FUNCTION_BLOCK FB_System_BSp_795
VAR_INPUT
	Freigabe_auto			: BOOL;
	Freigabe_Deakt_auto		: BOOL;
	Betrieb_Anford_auto		: BOOL;

	Regelung_Modus_auto		: SINT;
	Regelung_Sollw_auto		: REAL;

	Temp_Netz_KW			: REAL; (*Temperatur kommt aus den Netzen; setzt sich zusammen aus Temperatur der Pufferspeicher, dem Betonspeicher und der Umgebungstemperatur*)
END_VAR
VAR_OUTPUT
	{attribute 'OPC.UA.DA' := '1'}Steuerung				: ST_System_BSp_Steuerung;		
	{attribute 'OPC.UA.DA' := '1'}Stellwert				: ST_System_BSp_Stellwert;		
	{attribute 'OPC.UA.DA' := '1'}Zustand					: ST_System_BSp_Zustand;	
	{attribute 'OPC.UA.DA' := '1'}Parameter				: ST_System_BSp_Parameter;		
END_VAR
VAR
	Stellventil_105			: FB_SV;
	Pumpe_105				: FB_PU;
	Pumpe_710				: FB_PU_Schuetz;
	Betonspeicher_795		: FB_BSp;

	Zustandscheck			: FB_System_BSp_795_Zustandscheck;
	Logik					: FB_System_BSp_Logik;
	Ablaufsteuerung			: FB_System_BSp_Ablaufsteuerung;
	Sollwertscheck			: FB_System_BSp_Sollwertscheck;
	Stellwertscheck			: FB_System_BSp_Stellwertscheck;
	Regelung				: FB_System_BSp_Regelung;
	Temp_Bsp				: REAL;
END_VAR

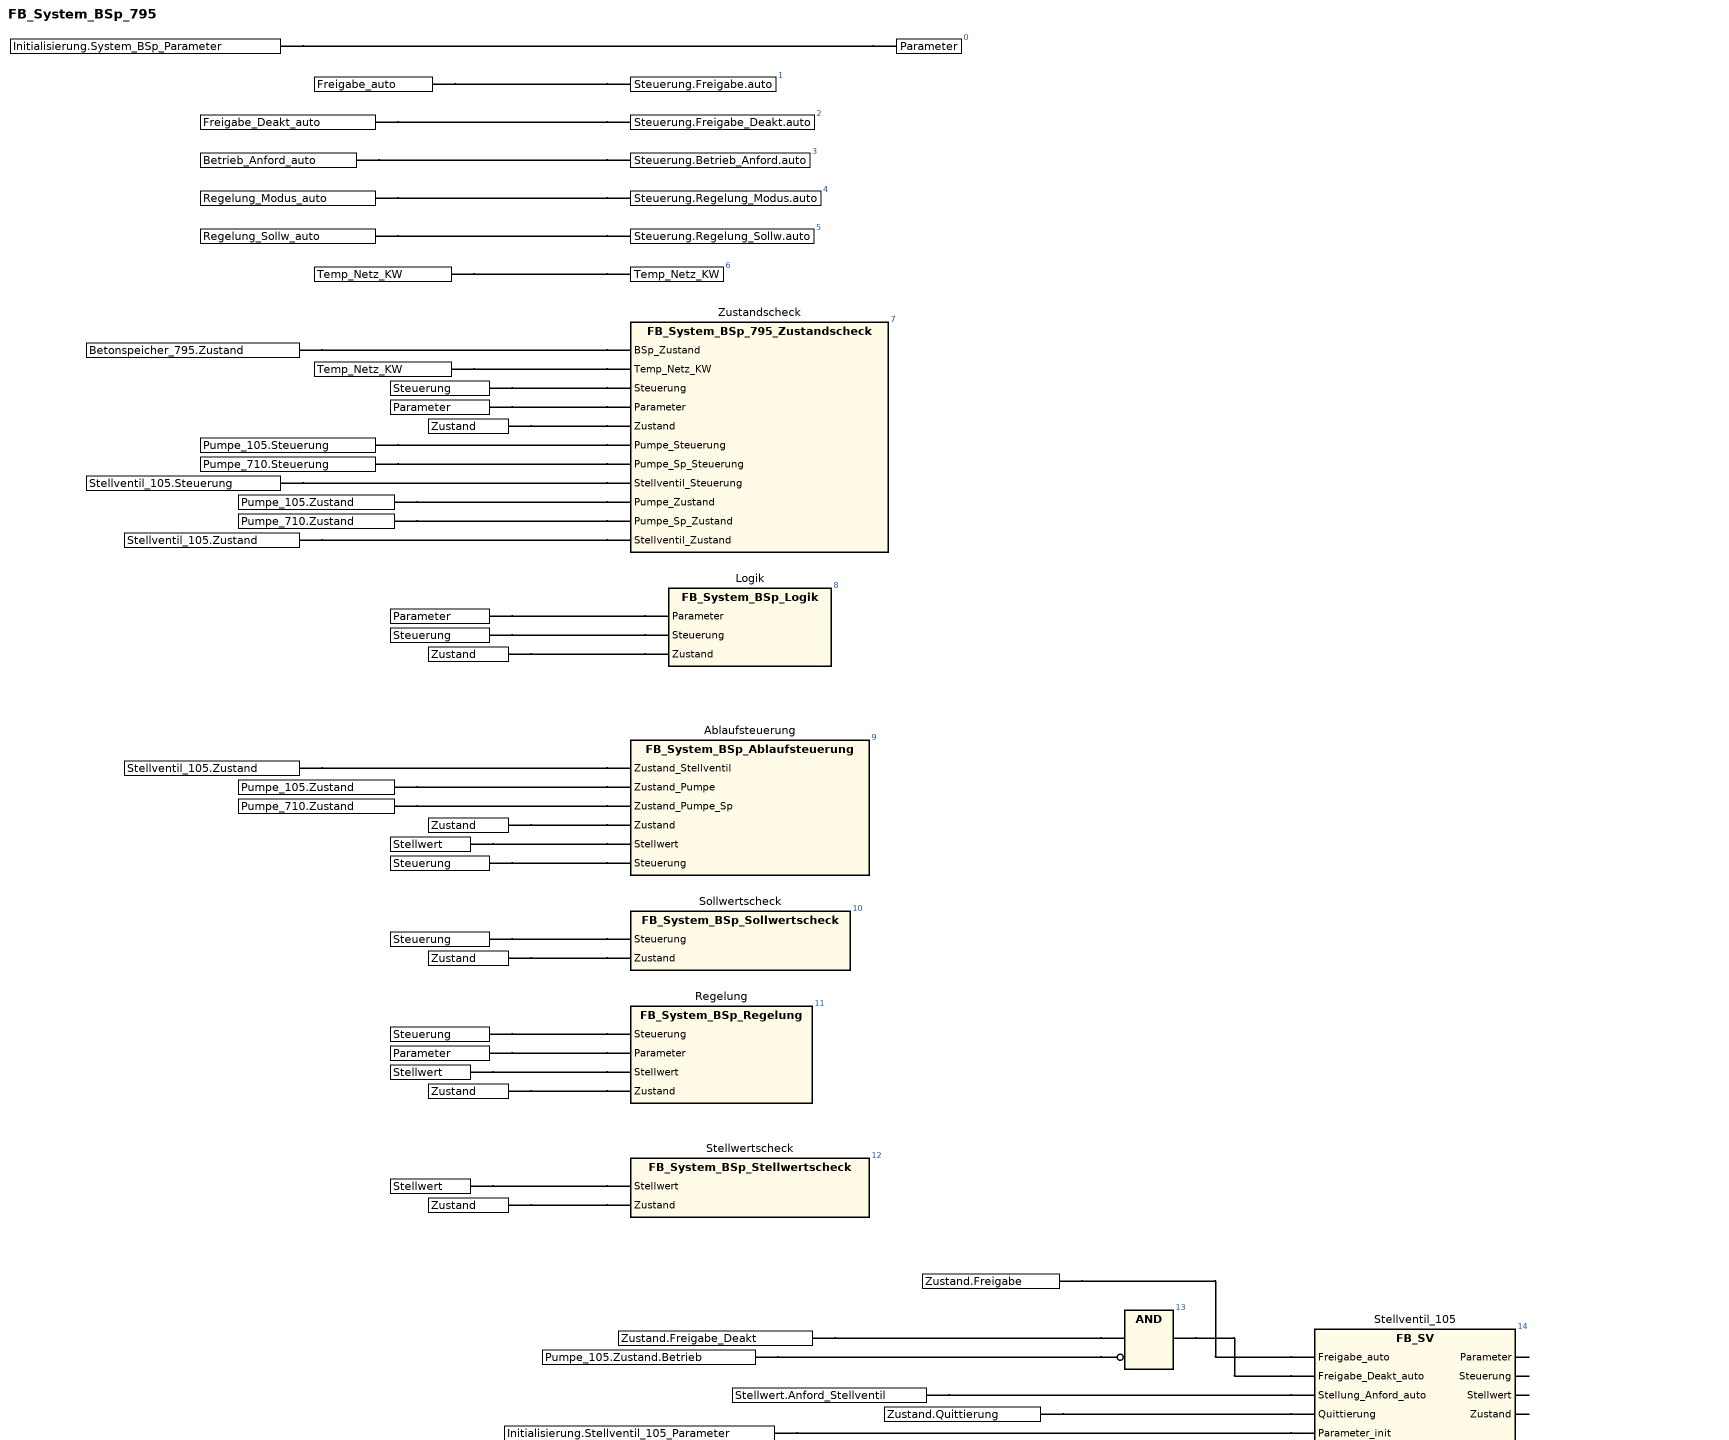
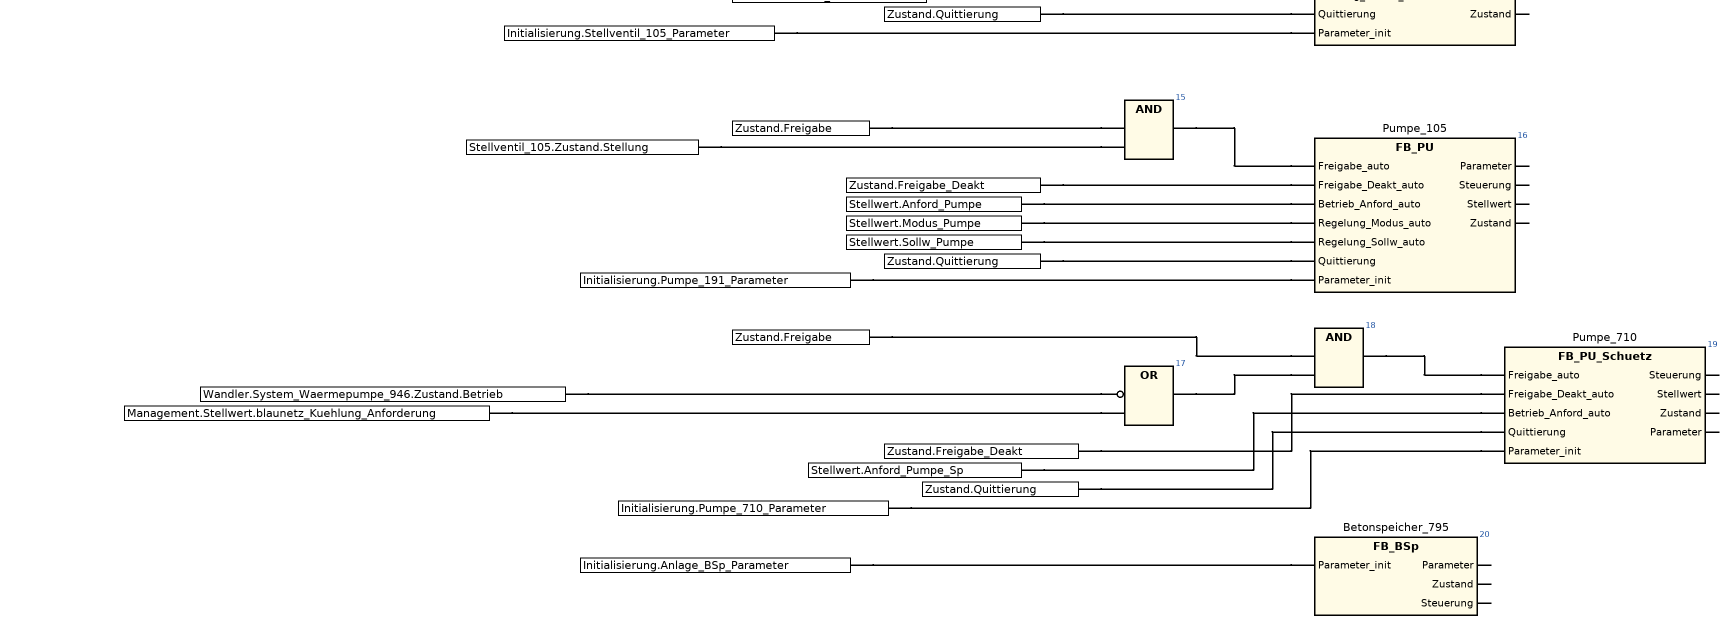
Parameter := Initialisierung.System_BSp_Parameter;
Steuerung.Freigabe.auto := Freigabe_auto;
Steuerung.Freigabe_Deakt.auto := Freigabe_Deakt_auto;
Steuerung.Betrieb_Anford.auto := Betrieb_Anford_auto;
Steuerung.Regelung_Modus.auto := Regelung_Modus_auto;
Steuerung.Regelung_Sollw.auto := Regelung_Sollw_auto;
Temp_Netz_KW := Temp_Netz_KW;
Zustandscheck(
    BSp_Zustand := Betonspeicher_795.Zustand,
    Temp_Netz_KW := Temp_Netz_KW,
    Steuerung := Steuerung,
    Parameter := Parameter,
    Zustand := Zustand,
    Pumpe_Steuerung := Pumpe_105.Steuerung,
    Pumpe_Sp_Steuerung := Pumpe_710.Steuerung,
    Stellventil_Steuerung := Stellventil_105.Steuerung,
    Pumpe_Zustand := Pumpe_105.Zustand,
    Pumpe_Sp_Zustand := Pumpe_710.Zustand,
    Stellventil_Zustand := Stellventil_105.Zustand); // FB_System_BSp_795_Zustandscheck
Logik(Parameter := Parameter, Steuerung := Steuerung, Zustand := Zustand); // FB_System_BSp_Logik
Ablaufsteuerung(
    Zustand_Stellventil := Stellventil_105.Zustand,
    Zustand_Pumpe := Pumpe_105.Zustand,
    Zustand_Pumpe_Sp := Pumpe_710.Zustand,
    Zustand := Zustand,
    Stellwert := Stellwert,
    Steuerung := Steuerung); // FB_System_BSp_Ablaufsteuerung
Sollwertscheck(Steuerung := Steuerung, Zustand := Zustand); // FB_System_BSp_Sollwertscheck
Regelung(Steuerung := Steuerung, Parameter := Parameter, Stellwert := Stellwert, Zustand := Zustand); // FB_System_BSp_Regelung
Stellwertscheck(Stellwert := Stellwert, Zustand := Zustand); // FB_System_BSp_Stellwertscheck
Stellventil_105(
    Freigabe_auto := Zustand.Freigabe,
    Freigabe_Deakt_auto := Zustand.Freigabe_Deakt AND NOT Pumpe_105.Zustand.Betrieb,
    Stellung_Anford_auto := Stellwert.Anford_Stellventil,
    Quittierung := Zustand.Quittierung,
    Parameter_init := Initialisierung.Stellventil_105_Parameter); // FB_SV
Pumpe_105(
    Freigabe_auto := Zustand.Freigabe AND Stellventil_105.Zustand.Stellung,
    Freigabe_Deakt_auto := Zustand.Freigabe_Deakt,
    Betrieb_Anford_auto := Stellwert.Anford_Pumpe,
    Regelung_Modus_auto := Stellwert.Modus_Pumpe,
    Regelung_Sollw_auto := Stellwert.Sollw_Pumpe,
    Quittierung := Zustand.Quittierung,
    Parameter_init := Initialisierung.Pumpe_191_Parameter); // FB_PU
Pumpe_710(
    Freigabe_auto := Zustand.Freigabe AND (NOT Wandler.System_Waermepumpe_946.Zustand.Betrieb OR Management.Stellwert.blaunetz_Kuehlung_Anforderung),
    Freigabe_Deakt_auto := Zustand.Freigabe_Deakt,
    Betrieb_Anford_auto := Stellwert.Anford_Pumpe_Sp,
    Quittierung := Zustand.Quittierung,
    Parameter_init := Initialisierung.Pumpe_710_Parameter); // FB_PU_Schuetz
Betonspeicher_795(Parameter_init := Initialisierung.Anlage_BSp_Parameter); // FB_BSp

END_FUNCTION_BLOCK

(* stored: Version 1.1.0.1, ProductVersion 3.1.4024.9
   POU FB_System_BSp_795: Id {bdbfd6dc-7825-463f-9aa4-f329050bec06}, SpecialFunc None *)
